FUNCTION_BLOCK SS2_ifb_Press (* Template for a Basic Function Block Type *)
  (* Standard: 61499-2 *)
  (* Version 1.0, 2024-07-25, DEVIASH *)
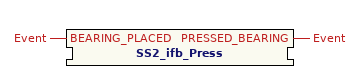
  EVENT_INPUT
    BEARING_PLACED; (* Initialization Request *)
  END_EVENT
  EVENT_OUTPUT
    PRESSED_BEARING; (* Initialization Confirm *)
  END_EVENT
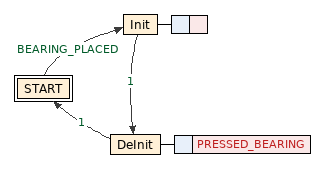
  EC_STATES
    START; (* Initial State *)
    Init; (* Initialization *)
    DeInit : -> PRESSED_BEARING;
  END_STATES
  EC_TRANSITIONS
    START TO Init := BEARING_PLACED;
    DeInit TO START := 1;
    Init TO DeInit := 1;
  END_TRANSITIONS
END_FUNCTION_BLOCK
